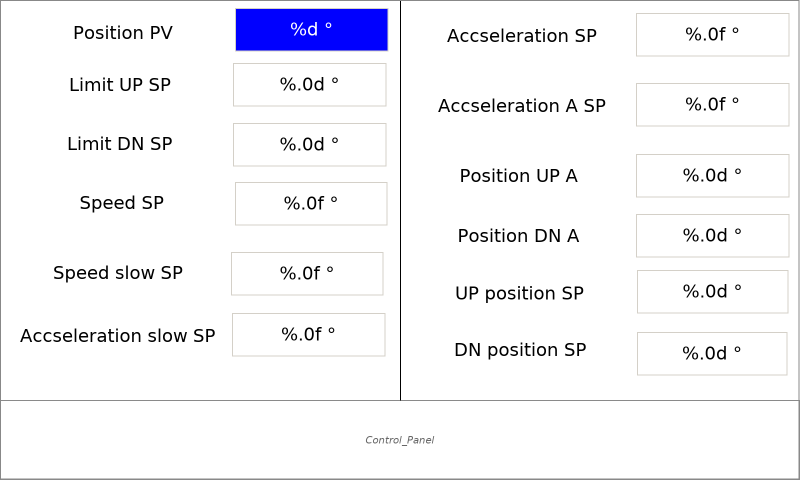
VISUALIZATION Settings  // 800x480
    Frame (0,400 800x80)
        shows Control_Panel()
    Textfield (636,154 153x43), "%.0d °", text variable: GVL_IO.Position_UP_A_SP
        OnMouseClick: write the text variable via Default
    Textfield (235,182 152x43), "%.0f °", text variable: GVL_IO.Speed_SP
        OnMouseClick: write the text variable via Default
    Label (20,18 206x30), "Position PV"
    Label (420,161 203x30), "Position UP A"
    Label (20,188 204x30), "Speed SP"
    Label (420,21 204x30), "Accseleration SP"
    Textfield (636,13 153x43), "%.0f °", text variable: GVL_IO.Accseleration_SP
        OnMouseClick: write the text variable via Default
    Textfield (235,8 153x43), "%d °", text variable: GVL_IO.Position_PV_HMI
    Label (17,70 206x30), "Limit UP SP"
    Textfield (233,63 153x43), "%.0d °", text variable: GVL_IO.Motor_Limit_UP
        OnMouseClick: write the text variable via Default
    Label (17,129 206x30), "Limit DN SP"
    Textfield (233,123 153x43), "%.0d °", text variable: GVL_IO.Motor_Limit_DN
        OnMouseClick: write the text variable via Default
    Line (400,0) (400,400)
    Label (420,221 203x30), "Position DN A"
    Textfield (636,214 153x43), "%.0d °", text variable: GVL_IO.Position_DN_A_SP
        OnMouseClick: write the text variable via Default
    Label (420,91 204x30), "Accseleration A SP"
    Textfield (636,83 153x43), "%.0f °", text variable: GVL_IO.Accseleration_A_SP
        OnMouseClick: write the text variable via Default
    Label (16,258 204x30), "Speed slow SP"
    Textfield (231,252 152x43), "%.0f °", text variable: GVL_IO.Speed_SP_slow
        OnMouseClick: write the text variable via Default
    Label (16,321 204x30), "Accseleration slow SP"
    Textfield (232,313 153x43), "%.0f °", text variable: GVL_IO.Accseleration_SP_slow
        OnMouseClick: write the text variable via Default
    Label (418,273 203x41), "UP position SP"
    Textfield (637,270 151x43), "%.0d °", text variable: GVL_IO.Position_UP_SP
        OnMouseClick: write the text variable via Default
    Label (403,325 235x50), "DN position SP"
    Textfield (637,332 150x43), "%.0d °", text variable: GVL_IO.Position_DN_SP
        OnMouseClick: write the text variable via Default
END_VISUALIZATION

(* stored: Version 1.1.0.1, ProductVersion 3.1.4024.13
   Visu Settings: Id {2934c60b-5318-4e55-b87c-3ba0e7ba11d7} *)
